// TIA Portal project "Pick & Place XYZ_V15.1" (V15.1)
// Vorlageprojekt für das Buch mit Zielsystem S7-1200

(* hardware
DEVICE "S7-1200-Station_1"  S7-1200 Station
   slot 0: "Baugruppenträger_0"  Rack  V1.0
   slot 1: "PLC_1"  CPU 1211C DC/DC/DC  6ES7 211-1AE40-0XB0  V4.1
*)

// ===== PLC "PLC_1"  CPU 1211C DC/DC/DC =====

VAR_GLOBAL   // PLC tag table "Standard-Variablentabelle"
   "Box at place" AT %I0.0 : Bool;
   "Part at place" AT %I0.1 : Bool;
   "Detected" AT %I0.2 : Bool;
   "C limit" AT %I0.3 : Bool;
   "Start" AT %I0.4 : Bool;
   "Reset" AT %I0.5 : Bool;
   "Stop" AT %I0.6 : Bool;
   "Emergency Stop" AT %I0.7 : Bool;
   "Auto" AT %I1.0 : Bool;
   "X" AT %ID30 : Real;
   "Y" AT %ID34 : Real;
   "Z" AT %ID38 : Real;
   "Box conveyor" AT %Q0.0 : Bool;
   "Part conveyor" AT %Q0.1 : Bool;
   "Exit conveyor" AT %Q0.2 : Bool;
   "C +" AT %Q0.3 : Bool;
   "Grab" AT %Q0.4 : Bool;
   "Exit green" AT %Q0.5 : Bool;
   "Exit yellow" AT %Q0.6 : Bool;
   "Exit red" AT %Q0.7 : Bool;
   "SP X" AT %QD30 : Real;
   "SP Y" AT %QD34 : Real;
   "SP Z" AT %QD38 : Real;
   "Counter" AT %QD42 : DInt;
   "Tag_1" AT %M100.0 : Bool;
   "Tag_2" AT %M100.1 : Bool;
   "Tag_3" AT %M100.2 : Bool;
   "Tag_5" AT %M100.4 : Bool;
   "Tag_6" AT %M100.5 : Bool;
   "Tag_10" AT %M101.1 : Bool;
   "Tag_4" AT %M100.3 : Bool;
   "Tag_7" AT %M100.6 : Bool;
END_VAR

VAR_GLOBAL   // PLC tag table "Default tag table"
   "Run" AT %M0.0 : Bool;
END_VAR

// folder: System blocks/Program resources

DATA_BLOCK "Counting_sp"   // DB1
{ S7_Optimized_Access := 'TRUE' }
AUTHOR : Simatic
FAMILY : IEC
NAME : CNTR
VERSION : 1.0
// stored: InstanceOfName IEC_COUNTER
"IEC_COUNTER"
BEGIN
END_DATA_BLOCK

// folder: (top level)

FUNCTION "Pick & Place XYZ" : Void   // FC1, LAD
{ S7_Optimized_Access := 'TRUE' }
VERSION : 0.1
   VAR_TEMP   // added for the SCL form of the ladder/FBD networks
      _w1 : Bool;
      _w2 : Bool;
   END_VAR
BEGIN

REGION Network 1: Box conveyor
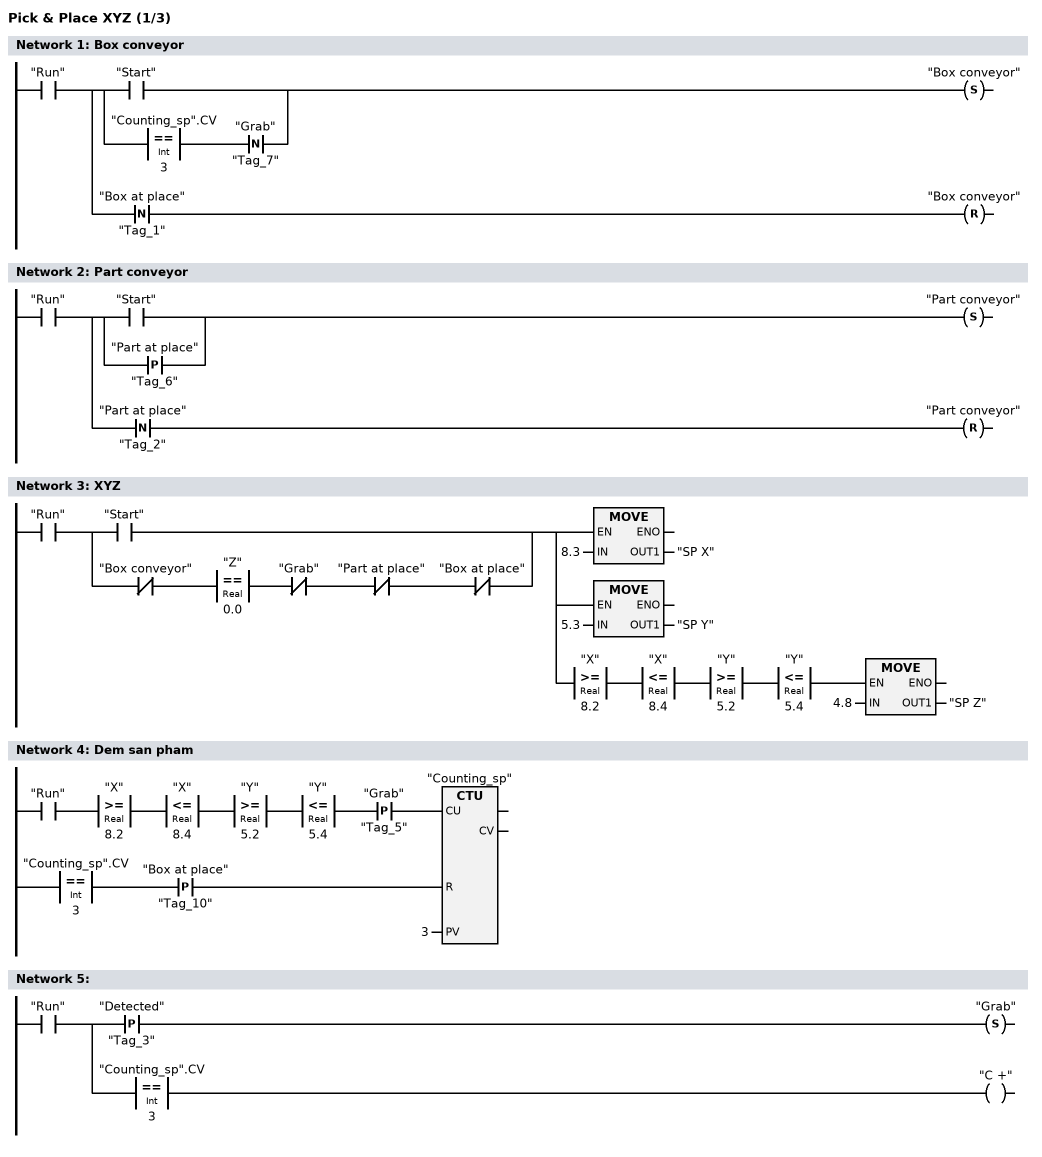
   RUNG wire#powerrail
      Contact( "Run" )
      wire#w1
      Contact( "Start" )
      wire#w2
      S_Coil( "Box conveyor" )
   END_RUNG
   RUNG wire#w1
      { S7_Templates := "SrcType := Int" } EQ_Contact(in1 := "Counting_sp".CV, in2 := 3)
      N_Contact(operand := "Grab", bit := "Tag_7")
   END_RUNG wire#w2
   RUNG wire#w1
      N_Contact(operand := "Box at place", bit := "Tag_1")
      R_Coil( "Box conveyor" )
   END_RUNG
   // the same network as SCL:
   #_w1 := "Run" AND ("Counting_sp".CV = 3) AND NOT "Grab" AND "Tag_7";   // falling edge of "Grab"
   "Tag_7" := "Grab";
   IF ("Run" AND "Start") OR #_w1 THEN "Box conveyor" := TRUE; END_IF;
   #_w2 := "Run" AND NOT "Box at place" AND "Tag_1";   // falling edge of "Box at place"
   "Tag_1" := "Box at place";
   IF #_w2 THEN "Box conveyor" := FALSE; END_IF;
END_REGION

REGION Network 2: Part conveyor
   RUNG wire#powerrail
      Contact( "Run" )
      wire#w1
      Contact( "Start" )
      wire#w2
      S_Coil( "Part conveyor" )
   END_RUNG
   RUNG wire#w1
      P_Contact(operand := "Part at place", bit := "Tag_6")
   END_RUNG wire#w2
   RUNG wire#w1
      N_Contact(operand := "Part at place", bit := "Tag_2")
      R_Coil( "Part conveyor" )
   END_RUNG
   // the same network as SCL:
   #_w1 := "Run" AND "Part at place" AND NOT "Tag_6";   // rising edge of "Part at place"
   "Tag_6" := "Part at place";
   IF ("Run" AND "Start") OR #_w1 THEN "Part conveyor" := TRUE; END_IF;
   #_w2 := "Run" AND NOT "Part at place" AND "Tag_2";   // falling edge of "Part at place"
   "Tag_2" := "Part at place";
   IF #_w2 THEN "Part conveyor" := FALSE; END_IF;
END_REGION

REGION Network 3: XYZ
   RUNG wire#powerrail
      Contact( "Run" )
      wire#w1
      Contact( "Start" )
      wire#w2
      Move(in := 8.3, out1 => "SP X")
   END_RUNG
   RUNG wire#w1
      I_Contact( "Box conveyor" )
      { S7_Templates := "SrcType := Real" } EQ_Contact(in1 := "Z", in2 := 0.0)
      I_Contact( "Grab" )
      I_Contact( "Part at place" )
      I_Contact( "Box at place" )
   END_RUNG wire#w2
   RUNG wire#w2
      Move(in := 5.3, out1 => "SP Y")
   END_RUNG
   RUNG wire#w2
      { S7_Templates := "SrcType := Real" } GE_Contact(in1 := "X", in2 := 8.2)
      { S7_Templates := "SrcType := Real" } LE_Contact(in1 := "X", in2 := 8.4)
      { S7_Templates := "SrcType := Real" } GE_Contact(in1 := "Y", in2 := 5.2)
      { S7_Templates := "SrcType := Real" } LE_Contact(in1 := "Y", in2 := 5.4)
      Move(in := 4.8, out1 => "SP Z")
   END_RUNG
   // the same network as SCL:
   #_w1 := "Run" AND ("Start" OR (NOT "Box conveyor" AND ("Z" = 0.0) AND NOT "Grab" AND NOT "Part at place" AND NOT "Box at place"));
   IF #_w1 THEN
       "SP X" := 8.3;
       "SP Y" := 5.3;
   END_IF;
   IF #_w1 AND ("X" >= 8.2) AND ("X" <= 8.4) AND ("Y" >= 5.2) AND ("Y" <= 5.4) THEN "SP Z" := 4.8; END_IF;
END_REGION

REGION Network 4: Dem san pham
   #_w1 := "Run" AND ("X" >= 8.2) AND ("X" <= 8.4) AND ("Y" >= 5.2) AND ("Y" <= 5.4) AND "Grab" AND NOT "Tag_5";   // rising edge of "Grab"
   "Tag_5" := "Grab";
   #_w2 := ("Counting_sp".CV = 3) AND "Box at place" AND NOT "Tag_10";   // rising edge of "Box at place"
   "Tag_10" := "Box at place";
   "Counting_sp".CTU(CU := #_w1, R := #_w2, PV := 3);
END_REGION

REGION Network 5
   RUNG wire#powerrail
      Contact( "Run" )
      wire#w1
      P_Contact(operand := "Detected", bit := "Tag_3")
      S_Coil( "Grab" )
   END_RUNG
   RUNG wire#w1
      { S7_Templates := "SrcType := Int" } EQ_Contact(in1 := "Counting_sp".CV, in2 := 3)
      Coil( "C +" )
   END_RUNG
   // the same network as SCL:
   #_w1 := "Run" AND "Detected" AND NOT "Tag_3";   // rising edge of "Detected"
   "Tag_3" := "Detected";
   IF #_w1 THEN "Grab" := TRUE; END_IF;
   "C +" := "Run" AND ("Counting_sp".CV = 3);
END_REGION

REGION Network 6: SP 1
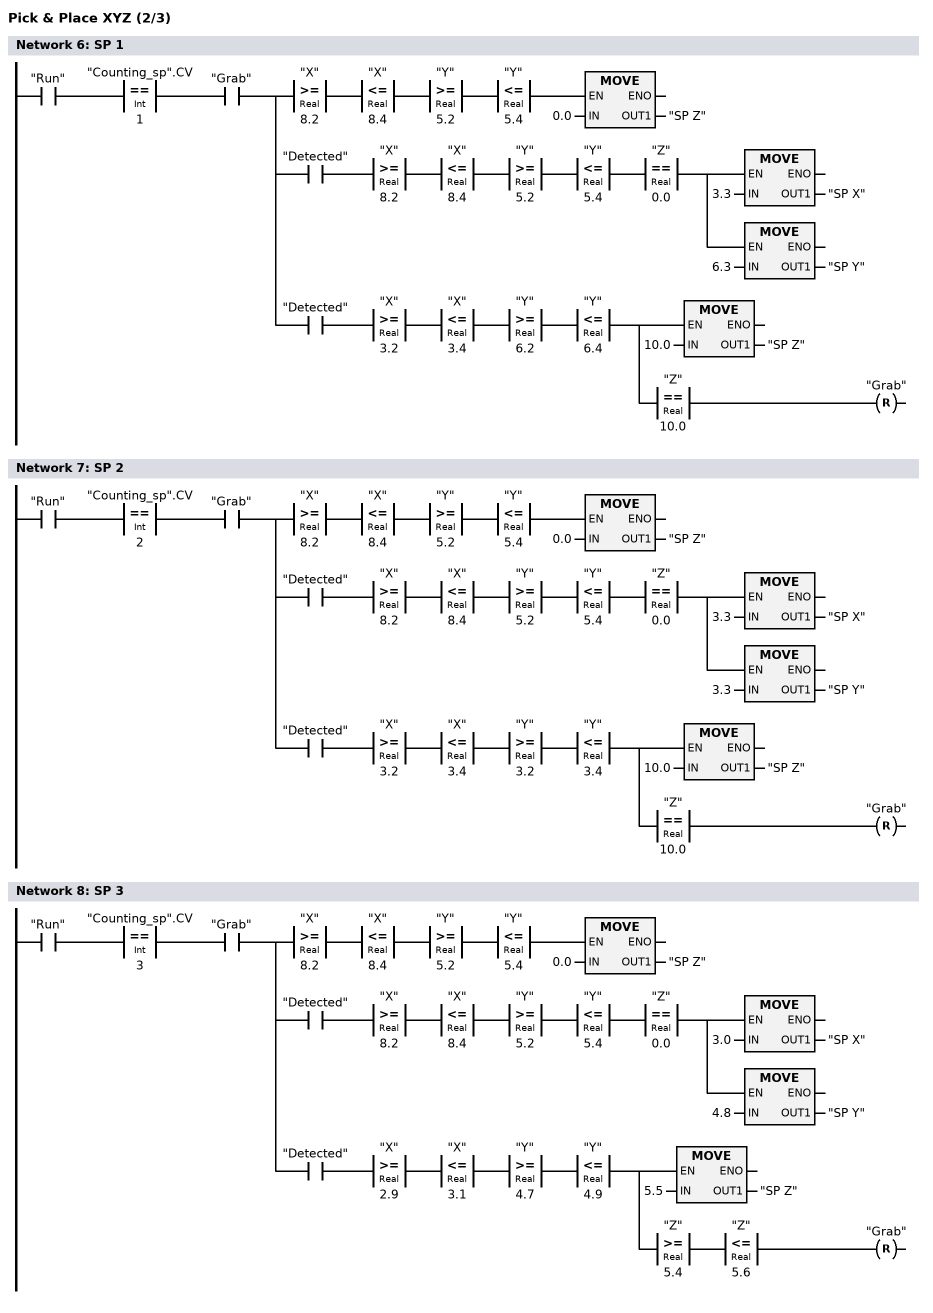
   RUNG wire#powerrail
      Contact( "Run" )
      { S7_Templates := "SrcType := Int" } EQ_Contact(in1 := "Counting_sp".CV, in2 := 1)
      Contact( "Grab" )
      wire#w1
      { S7_Templates := "SrcType := Real" } GE_Contact(in1 := "X", in2 := 8.2)
      { S7_Templates := "SrcType := Real" } LE_Contact(in1 := "X", in2 := 8.4)
      { S7_Templates := "SrcType := Real" } GE_Contact(in1 := "Y", in2 := 5.2)
      { S7_Templates := "SrcType := Real" } LE_Contact(in1 := "Y", in2 := 5.4)
      Move(in := 0.0, out1 => "SP Z")
   END_RUNG
   RUNG wire#w1
      Contact( "Detected" )
      { S7_Templates := "SrcType := Real" } GE_Contact(in1 := "X", in2 := 8.2)
      { S7_Templates := "SrcType := Real" } LE_Contact(in1 := "X", in2 := 8.4)
      { S7_Templates := "SrcType := Real" } GE_Contact(in1 := "Y", in2 := 5.2)
      { S7_Templates := "SrcType := Real" } LE_Contact(in1 := "Y", in2 := 5.4)
      { S7_Templates := "SrcType := Real" } EQ_Contact(in1 := "Z", in2 := 0.0)
      wire#w2
      Move(in := 3.3, out1 => "SP X")
   END_RUNG
   RUNG wire#w2
      Move(in := 6.3, out1 => "SP Y")
   END_RUNG
   RUNG wire#w1
      Contact( "Detected" )
      { S7_Templates := "SrcType := Real" } GE_Contact(in1 := "X", in2 := 3.2)
      { S7_Templates := "SrcType := Real" } LE_Contact(in1 := "X", in2 := 3.4)
      { S7_Templates := "SrcType := Real" } GE_Contact(in1 := "Y", in2 := 6.2)
      { S7_Templates := "SrcType := Real" } LE_Contact(in1 := "Y", in2 := 6.4)
      wire#w3
      Move(in := 10.0, out1 => "SP Z")
   END_RUNG
   RUNG wire#w3
      { S7_Templates := "SrcType := Real" } EQ_Contact(in1 := "Z", in2 := 10.0)
      R_Coil( "Grab" )
   END_RUNG
   // the same network as SCL:
   #_w1 := "Run" AND ("Counting_sp".CV = 1) AND "Grab";
   IF #_w1 AND ("X" >= 8.2) AND ("X" <= 8.4) AND ("Y" >= 5.2) AND ("Y" <= 5.4) THEN "SP Z" := 0.0; END_IF;
   IF #_w1 AND "Detected" AND ("X" >= 8.2) AND ("X" <= 8.4) AND ("Y" >= 5.2) AND ("Y" <= 5.4) AND ("Z" = 0.0) THEN
       "SP X" := 3.3;
       "SP Y" := 6.3;
   END_IF;
   #_w2 := #_w1 AND "Detected" AND ("X" >= 3.2) AND ("X" <= 3.4) AND ("Y" >= 6.2) AND ("Y" <= 6.4);
   IF #_w2 THEN "SP Z" := 10.0; END_IF;
   IF #_w2 AND ("Z" = 10.0) THEN "Grab" := FALSE; END_IF;
END_REGION

REGION Network 7: SP 2
   RUNG wire#powerrail
      Contact( "Run" )
      { S7_Templates := "SrcType := Int" } EQ_Contact(in1 := "Counting_sp".CV, in2 := 2)
      Contact( "Grab" )
      wire#w1
      { S7_Templates := "SrcType := Real" } GE_Contact(in1 := "X", in2 := 8.2)
      { S7_Templates := "SrcType := Real" } LE_Contact(in1 := "X", in2 := 8.4)
      { S7_Templates := "SrcType := Real" } GE_Contact(in1 := "Y", in2 := 5.2)
      { S7_Templates := "SrcType := Real" } LE_Contact(in1 := "Y", in2 := 5.4)
      Move(in := 0.0, out1 => "SP Z")
   END_RUNG
   RUNG wire#w1
      Contact( "Detected" )
      { S7_Templates := "SrcType := Real" } GE_Contact(in1 := "X", in2 := 8.2)
      { S7_Templates := "SrcType := Real" } LE_Contact(in1 := "X", in2 := 8.4)
      { S7_Templates := "SrcType := Real" } GE_Contact(in1 := "Y", in2 := 5.2)
      { S7_Templates := "SrcType := Real" } LE_Contact(in1 := "Y", in2 := 5.4)
      { S7_Templates := "SrcType := Real" } EQ_Contact(in1 := "Z", in2 := 0.0)
      wire#w2
      Move(in := 3.3, out1 => "SP X")
   END_RUNG
   RUNG wire#w2
      Move(in := 3.3, out1 => "SP Y")
   END_RUNG
   RUNG wire#w1
      Contact( "Detected" )
      { S7_Templates := "SrcType := Real" } GE_Contact(in1 := "X", in2 := 3.2)
      { S7_Templates := "SrcType := Real" } LE_Contact(in1 := "X", in2 := 3.4)
      { S7_Templates := "SrcType := Real" } GE_Contact(in1 := "Y", in2 := 3.2)
      { S7_Templates := "SrcType := Real" } LE_Contact(in1 := "Y", in2 := 3.4)
      wire#w3
      Move(in := 10.0, out1 => "SP Z")
   END_RUNG
   RUNG wire#w3
      { S7_Templates := "SrcType := Real" } EQ_Contact(in1 := "Z", in2 := 10.0)
      R_Coil( "Grab" )
   END_RUNG
   // the same network as SCL:
   #_w1 := "Run" AND ("Counting_sp".CV = 2) AND "Grab";
   IF #_w1 AND ("X" >= 8.2) AND ("X" <= 8.4) AND ("Y" >= 5.2) AND ("Y" <= 5.4) THEN "SP Z" := 0.0; END_IF;
   IF #_w1 AND "Detected" AND ("X" >= 8.2) AND ("X" <= 8.4) AND ("Y" >= 5.2) AND ("Y" <= 5.4) AND ("Z" = 0.0) THEN
       "SP X" := 3.3;
       "SP Y" := 3.3;
   END_IF;
   #_w2 := #_w1 AND "Detected" AND ("X" >= 3.2) AND ("X" <= 3.4) AND ("Y" >= 3.2) AND ("Y" <= 3.4);
   IF #_w2 THEN "SP Z" := 10.0; END_IF;
   IF #_w2 AND ("Z" = 10.0) THEN "Grab" := FALSE; END_IF;
END_REGION

REGION Network 8: SP 3
   RUNG wire#powerrail
      Contact( "Run" )
      { S7_Templates := "SrcType := Int" } EQ_Contact(in1 := "Counting_sp".CV, in2 := 3)
      Contact( "Grab" )
      wire#w1
      { S7_Templates := "SrcType := Real" } GE_Contact(in1 := "X", in2 := 8.2)
      { S7_Templates := "SrcType := Real" } LE_Contact(in1 := "X", in2 := 8.4)
      { S7_Templates := "SrcType := Real" } GE_Contact(in1 := "Y", in2 := 5.2)
      { S7_Templates := "SrcType := Real" } LE_Contact(in1 := "Y", in2 := 5.4)
      Move(in := 0.0, out1 => "SP Z")
   END_RUNG
   RUNG wire#w1
      Contact( "Detected" )
      { S7_Templates := "SrcType := Real" } GE_Contact(in1 := "X", in2 := 8.2)
      { S7_Templates := "SrcType := Real" } LE_Contact(in1 := "X", in2 := 8.4)
      { S7_Templates := "SrcType := Real" } GE_Contact(in1 := "Y", in2 := 5.2)
      { S7_Templates := "SrcType := Real" } LE_Contact(in1 := "Y", in2 := 5.4)
      { S7_Templates := "SrcType := Real" } EQ_Contact(in1 := "Z", in2 := 0.0)
      wire#w2
      Move(in := 3.0, out1 => "SP X")
   END_RUNG
   RUNG wire#w2
      Move(in := 4.8, out1 => "SP Y")
   END_RUNG
   RUNG wire#w1
      Contact( "Detected" )
      { S7_Templates := "SrcType := Real" } GE_Contact(in1 := "X", in2 := 2.9)
      { S7_Templates := "SrcType := Real" } LE_Contact(in1 := "X", in2 := 3.1)
      { S7_Templates := "SrcType := Real" } GE_Contact(in1 := "Y", in2 := 4.7)
      { S7_Templates := "SrcType := Real" } LE_Contact(in1 := "Y", in2 := 4.9)
      wire#w3
      Move(in := 5.5, out1 => "SP Z")
   END_RUNG
   RUNG wire#w3
      { S7_Templates := "SrcType := Real" } GE_Contact(in1 := "Z", in2 := 5.4)
      { S7_Templates := "SrcType := Real" } LE_Contact(in1 := "Z", in2 := 5.6)
      R_Coil( "Grab" )
   END_RUNG
   // the same network as SCL:
   #_w1 := "Run" AND ("Counting_sp".CV = 3) AND "Grab";
   IF #_w1 AND ("X" >= 8.2) AND ("X" <= 8.4) AND ("Y" >= 5.2) AND ("Y" <= 5.4) THEN "SP Z" := 0.0; END_IF;
   IF #_w1 AND "Detected" AND ("X" >= 8.2) AND ("X" <= 8.4) AND ("Y" >= 5.2) AND ("Y" <= 5.4) AND ("Z" = 0.0) THEN
       "SP X" := 3.0;
       "SP Y" := 4.8;
   END_IF;
   #_w2 := #_w1 AND "Detected" AND ("X" >= 2.9) AND ("X" <= 3.1) AND ("Y" >= 4.7) AND ("Y" <= 4.9);
   IF #_w2 THEN "SP Z" := 5.5; END_IF;
   IF #_w2 AND ("Z" >= 5.4) AND ("Z" <= 5.6) THEN "Grab" := FALSE; END_IF;
END_REGION

REGION Network 9
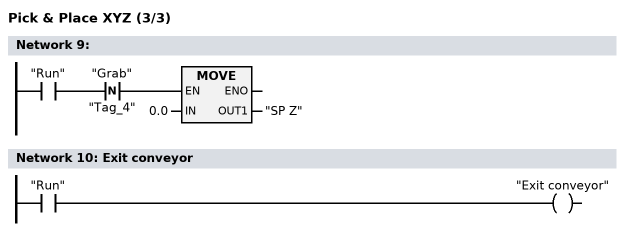
   RUNG wire#powerrail
      Contact( "Run" )
      N_Contact(operand := "Grab", bit := "Tag_4")
      Move(in := 0.0, out1 => "SP Z")
   END_RUNG
   // the same network as SCL:
   #_w1 := "Run" AND NOT "Grab" AND "Tag_4";   // falling edge of "Grab"
   "Tag_4" := "Grab";
   IF #_w1 THEN "SP Z" := 0.0; END_IF;
END_REGION

REGION Network 10: Exit conveyor
   RUNG wire#powerrail
      Contact( "Run" )
      Coil( "Exit conveyor" )
   END_RUNG
   // the same network as SCL:
   "Exit conveyor" := "Run";
END_REGION
END_FUNCTION

FUNCTION "MHJ-PLC-Lab-Function-S71200" : Void   // FC9000, SCL
{ S7_Optimized_Access := 'TRUE' }
VERSION : 0.1
   VAR_TEMP
      rdTimeReturn : Int;
      outputTime : DTL;
      SyncVal : Byte;
      forVal : Int;
      forVal_2 : Int;
      Value : Byte;
   END_VAR
   VAR CONSTANT
      CompVal : Byte := 16#34;
      Value_01 : Byte := 16#11;
      Value_01_DW : DWord := 16#A165_D992;
      Value_02_DW : DWord := 16#58BE_4401;
   END_VAR
BEGIN

   #Value:=PEEK(area := 16#82,
        dbNumber := 0,
        byteOffset := 511);
   #Value := #Value + 1;

   POKE(area := 16#82,
        dbNumber := 0,
        byteOffset := 511,
        value := #Value);

   POKE(area:=16#81,
        dbNumber:=0,
        byteOffset:=1016,
        value:=#Value_01_DW);
   POKE(area := 16#81,
        dbNumber := 0,
        byteOffset := 1020,
        value := #Value_02_DW);

   POKE(area := 16#81,
        dbNumber := 0,
        byteOffset := 511,
        value := B#16#00);

   FOR #forVal := 0 TO 120 DO
       FOR #forVal_2:=0 TO 10 DO
           #rdTimeReturn:=RD_SYS_T(#outputTime);
           #rdTimeReturn := WR_SYS_T(#outputTime);
           #rdTimeReturn := RD_SYS_T(#outputTime);
           #rdTimeReturn := WR_SYS_T(#outputTime);
       END_FOR;
       #SyncVal:= PEEK(area := 16#81,
                      dbNumber := 0,
                      byteOffset := 511);
       IF #SyncVal = #CompVal THEN
          GOTO M_1;
       END_IF;
   END_FOR;
   RETURN;

   M_1:
   POKE(area := 16#81,
        dbNumber := 0,
        byteOffset := 511,
        value := B#16#0);
END_FUNCTION

ORGANIZATION_BLOCK "Main"   // OB1, LAD, ProgramCycle
TITLE = "Main Program Sweep (Cycle)"
{ S7_Optimized_Access := 'TRUE' }
VERSION : 0.1
   VAR_INPUT
      Initial_Call : Bool;   // Initial call of this OB
      Remanence : Bool;   // =True, if remanent data are available
   END_VAR
BEGIN

REGION Network 1: Connection block for PLCSIM communications. Don't delete this network!
   // Im Netzwerk 1 wird der Konnektierungsbaustein für PLC-Lab aufgerufen.
   // Dieser Aufruf darf nicht entfernt werden!
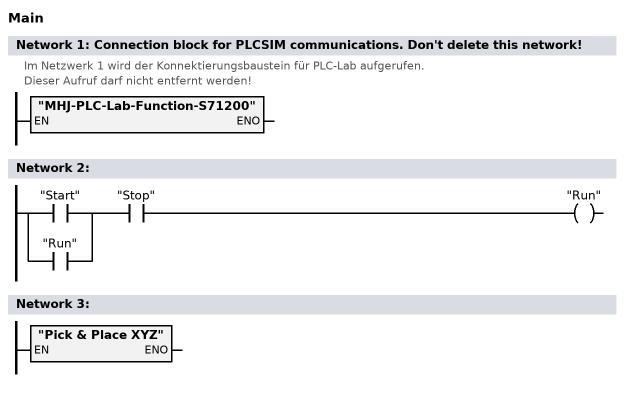
   RUNG wire#powerrail
      "MHJ-PLC-Lab-Function-S71200"()
   END_RUNG
   // the same network as SCL:
   "MHJ-PLC-Lab-Function-S71200"();
END_REGION

REGION Network 2
   RUNG wire#powerrail
      Contact( "Start" )
      wire#w1
      Contact( "Stop" )
      Coil( "Run" )
   END_RUNG
   RUNG wire#powerrail
      Contact( "Run" )
   END_RUNG wire#w1
   // the same network as SCL:
   "Run" := ("Start" OR "Run") AND "Stop";
END_REGION

REGION Network 3
   RUNG wire#powerrail
      "Pick & Place XYZ"()
   END_RUNG
   // the same network as SCL:
   "Pick & Place XYZ"();
END_REGION
END_ORGANIZATION_BLOCK